INTERFACE I_TimeProvider

PROPERTY TimestampMs : ULINT
GET
END_GET
END_PROPERTY

END_INTERFACE

(* stored: Version 1.1.0.1, ProductVersion 3.1.4024.12
   Itf I_TimeProvider: Id {eb4530fd-c524-05d3-19c5-8a230be0c1f5}
   Property TimestampMs: Id {09385750-0c1a-05bc-35ae-8131e2c24181}
   Get Get: Id {bc43b595-ae40-0665-31ac-9af7e97594c8} *)
